TYPE E_OperationMode : (
    OP_MODE_INVALID := 0,
    OP_MODE_MAINTENANCE := 10,
    OP_MODE_MANUAL := 20,
    OP_MODE_AUTOMATIC := 30
); END_TYPE

(* stored: Version 1.1.0.1
   DUT E_OperationMode: Id {E3000000-0000-4000-8000-000000000001} *)
